# EPICS substitutions: TPGSup/TPG300_function_statuses_error_setter.substitutions
file $(UTILITIES)/db/error_setter.template {

pattern {P, STREAM_PV, PV_NAME}
 {"\$(P)", "FUNCTION:STATUS:RB", "FUNCTION:STATUS:1:RB"}
 {"\$(P)", "FUNCTION:STATUS:RB", "FUNCTION:STATUS:2:RB"}
 {"\$(P)", "FUNCTION:STATUS:RB", "FUNCTION:STATUS:3:RB"}
 {"\$(P)", "FUNCTION:STATUS:RB", "FUNCTION:STATUS:4:RB"}

}
